% RSLogix 500 project BESTANDMANAGEMENT.RSS, saved by version 8.30.00.16 %
PROJECT "UNTITLED"    % processor: Bul.1763 MicroLogix 1100 Series B %

PROGRAM FILES
  LAD 2 "MAIN"  5 rungs
  LAD 3 "REIFEN"  5 rungs
  LAD 4 "FELGEN"  5 rungs
  LAD 5 "STOßDÄMPFE"  5 rungs

DATA FILES
  O0 OUTPUT  4 elements
  I1 INPUT  6 elements
  S2 STATUS  66 elements
  B3 BINARY  1 elements
  T4 TIMER  1 elements
  C5 COUNTER  1 elements
  R6 CONTROL  1 elements
  N7 INTEGER  9 elements
  F8 FLOAT  1 elements
  ST9 STRING  13 elements

LADDER 2 "MAIN"
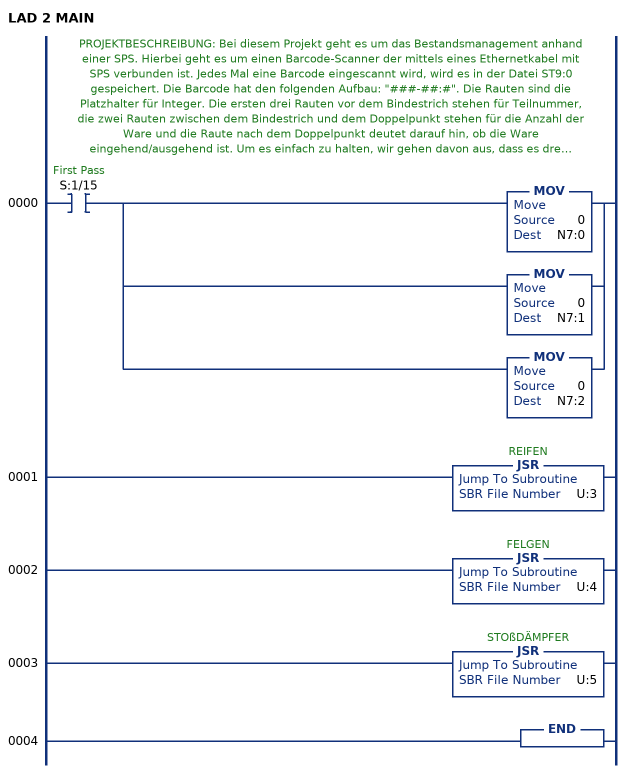
% Rung: 0 %
% PROJEKTBESCHREIBUNG: Bei diesem Projekt geht es um das Bestandsmanagement anhand einer SPS. Hierbei geht es um einen Barcode-Scanner der mittels eines Ethernetkabel mit SPS verbunden ist. Jedes Mal eine Barcode eingescannt wird, wird es in der Datei ST9:0 gespeichert. Die Barcode hat den folgenden Aufbau: "###-##:#". Die Rauten sind die Platzhalter für Integer. Die ersten drei Rauten vor dem Bindestrich stehen für Teilnummer, die zwei Rauten zwischen dem Bindestrich und dem Doppelpunkt stehen für die Anzahl der Ware und die Raute nach dem Doppelpunkt deutet darauf hin, ob die Ware eingehend/ausgehend ist. Um es einfach zu halten, wir gehen davon aus, dass es drei verschiedene Teile verwaltet werden. Teilnummer eins sind die Reifen mit der Teilnummer 123 , Teilnummer zwei sind die Felgen mit der Teilnummer 456 und Teilnummer drei sind die Stoßdämpfer mit der Nummer 789. Die letze Raute ist 1 beim Wareneingang und 2 beim Warenausgang.  N7:0 speichert die Anzahl der Reifen, N7:1 speichert die Anzahl der Felgen und N7:2 speichert die Anzahl der Stoßdämpfer. Beim Initialisierung wird sichergestellt, dass der Lager leer ist. %
SOR XIC S:1/15 BST MOV 0 N7:0 NXB MOV 0 N7:1 NXB MOV 0 N7:2 BND EOR
%   S:1/15  "First Pass" %
% Rung: 1 %
SOR JSR U:3 EOR
%   U:3  "REIFEN" %
% Rung: 2 %
SOR JSR U:4 EOR
%   U:4  "FELGEN" %
% Rung: 3 %
SOR JSR U:5 EOR
%   U:5  "STOßDÄMPFER" %
% Rung: 4 %
SOR END EOR

LADDER 3 "REIFEN"
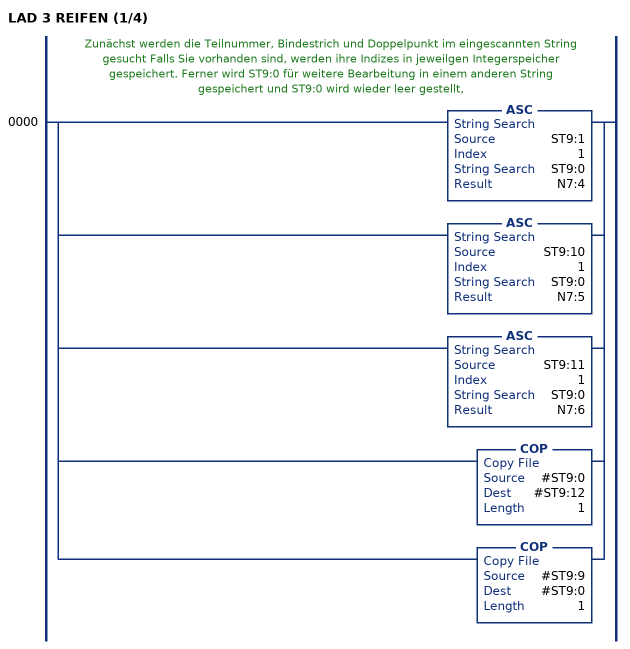
% Rung: 0 %
% Zunächst werden die Teilnummer, Bindestrich und Doppelpunkt im eingescannten String gesucht Falls Sie vorhanden sind, werden ihre Indizes in jeweilgen Integerspeicher gespeichert. Ferner wird ST9:0 für weitere Bearbeitung in einem anderen String gespeichert und ST9:0 wird wieder leer gestellt, %
SOR BST ASC ST9:1 1 ST9:0 N7:4 NXB ASC ST9:10 1 ST9:0 N7:5 NXB ASC ST9:11 1 ST9:0 N7:6 NXB COP #ST9:0 #ST9:12 1 NXB COP #ST9:9 #ST9:0 1 BND EOR
%   N7:4  "Index von Reifennummer" %
%   N7:5  "Index von Bindestrich" %
%   N7:6  "Index von Doppelpunkt" %

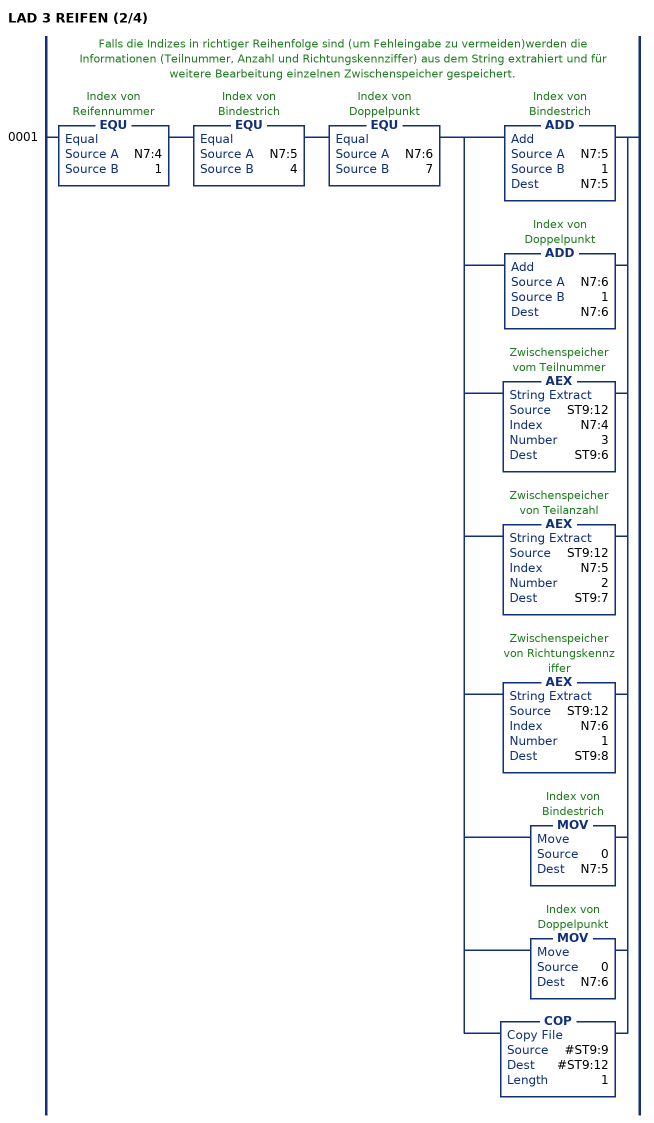
% Rung: 1 %
% Falls die Indizes in richtiger Reihenfolge sind (um Fehleingabe zu vermeiden)werden die Informationen (Teilnummer, Anzahl und Richtungskennziffer) aus dem String extrahiert und für weitere Bearbeitung einzelnen Zwischenspeicher gespeichert. %
SOR EQU N7:4 1 EQU N7:5 4 EQU N7:6 7 BST ADD N7:5 1 N7:5 NXB ADD N7:6 1 N7:6 NXB AEX ST9:12 N7:4 3 ST9:6 NXB AEX ST9:12 N7:5 2 ST9:7 NXB AEX ST9:12 N7:6 1 ST9:8 NXB MOV 0 N7:5 NXB MOV 0 N7:6 NXB COP #ST9:9 #ST9:12 1 BND EOR
%   N7:4  "Index von Reifennummer" %
%   N7:5  "Index von Bindestrich" %
%   N7:6  "Index von Doppelpunkt" %
%   ST9:6  "Zwischenspeicher vom Teilnummer" %
%   ST9:7  "Zwischenspeicher von Teilanzahl" %
%   ST9:8  "Zwischenspeicher von Richtungskennziffer" %

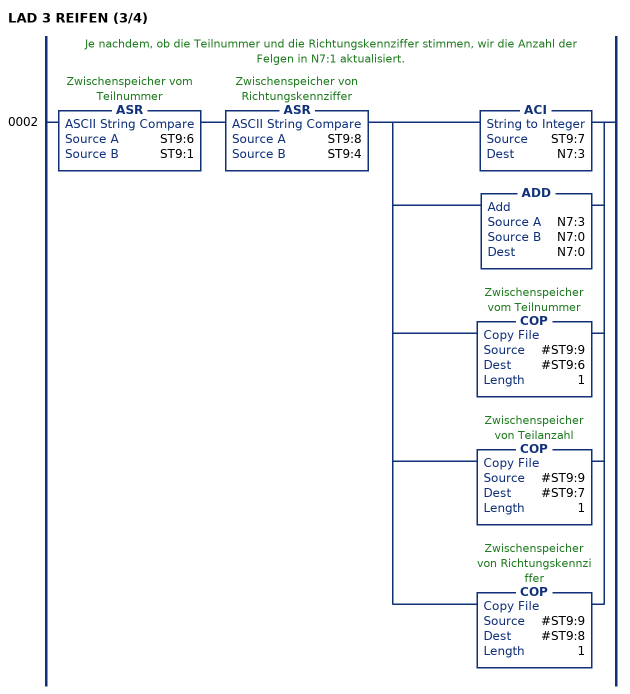
% Rung: 2 %
% Je nachdem, ob die Teilnummer und die Richtungskennziffer stimmen, wir die Anzahl der Felgen in N7:1 aktualisiert. %
SOR ASR ST9:6 ST9:1 ASR ST9:8 ST9:4 BST ACI ST9:7 N7:3 NXB ADD N7:3 N7:0 N7:0 NXB COP #ST9:9 #ST9:6 1 NXB COP #ST9:9 #ST9:7 1 NXB COP #ST9:9 #ST9:8 1 BND EOR
%   ST9:6  "Zwischenspeicher vom Teilnummer" %
%   ST9:8  "Zwischenspeicher von Richtungskennziffer" %
%   ST9:7  "Zwischenspeicher von Teilanzahl" %

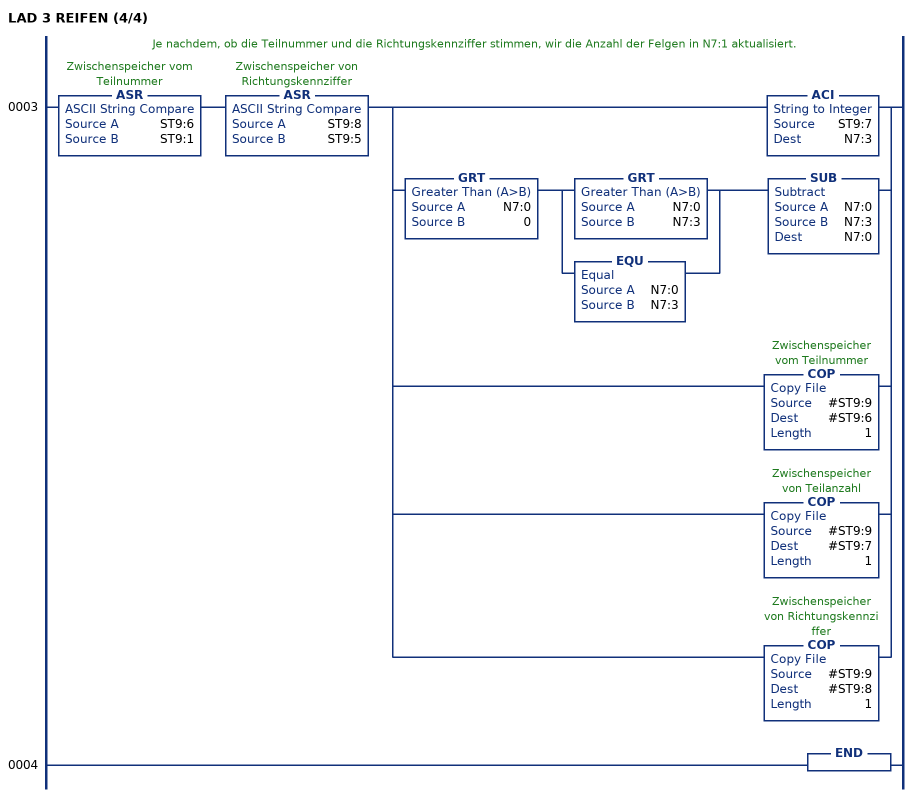
% Rung: 3 %
% Je nachdem, ob die Teilnummer und die Richtungskennziffer stimmen, wir die Anzahl der Felgen in N7:1 aktualisiert. %
SOR ASR ST9:6 ST9:1 ASR ST9:8 ST9:5 BST ACI ST9:7 N7:3 NXB GRT N7:0 0 BST GRT N7:0 N7:3 NXB EQU N7:0 N7:3 BND SUB N7:0 N7:3 N7:0 NXB COP #ST9:9 #ST9:6 1 NXB COP #ST9:9 #ST9:7 1 NXB COP #ST9:9 #ST9:8 1 BND EOR
%   ST9:6  "Zwischenspeicher vom Teilnummer" %
%   ST9:8  "Zwischenspeicher von Richtungskennziffer" %
%   ST9:7  "Zwischenspeicher von Teilanzahl" %
% Rung: 4 %
SOR END EOR

LADDER 4 "FELGEN"
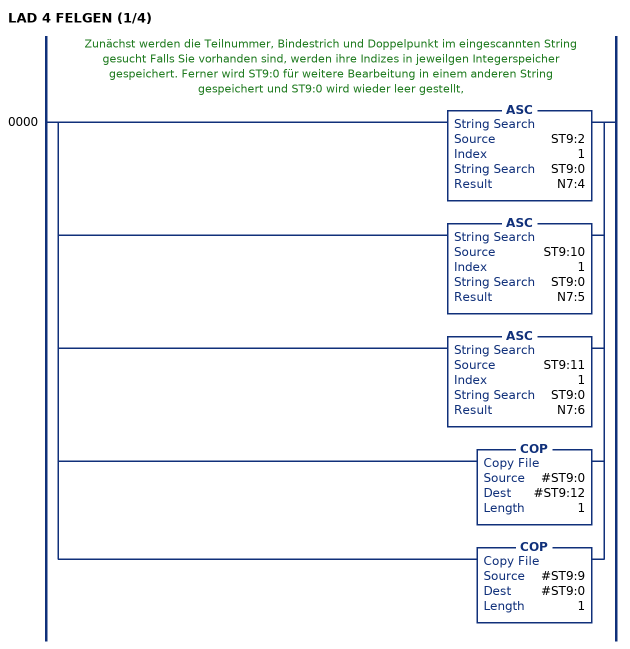
% Rung: 0 %
% Zunächst werden die Teilnummer, Bindestrich und Doppelpunkt im eingescannten String gesucht Falls Sie vorhanden sind, werden ihre Indizes in jeweilgen Integerspeicher gespeichert. Ferner wird ST9:0 für weitere Bearbeitung in einem anderen String gespeichert und ST9:0 wird wieder leer gestellt, %
SOR BST ASC ST9:2 1 ST9:0 N7:4 NXB ASC ST9:10 1 ST9:0 N7:5 NXB ASC ST9:11 1 ST9:0 N7:6 NXB COP #ST9:0 #ST9:12 1 NXB COP #ST9:9 #ST9:0 1 BND EOR
%   N7:4  "Index von Reifennummer" %
%   N7:5  "Index von Bindestrich" %
%   N7:6  "Index von Doppelpunkt" %

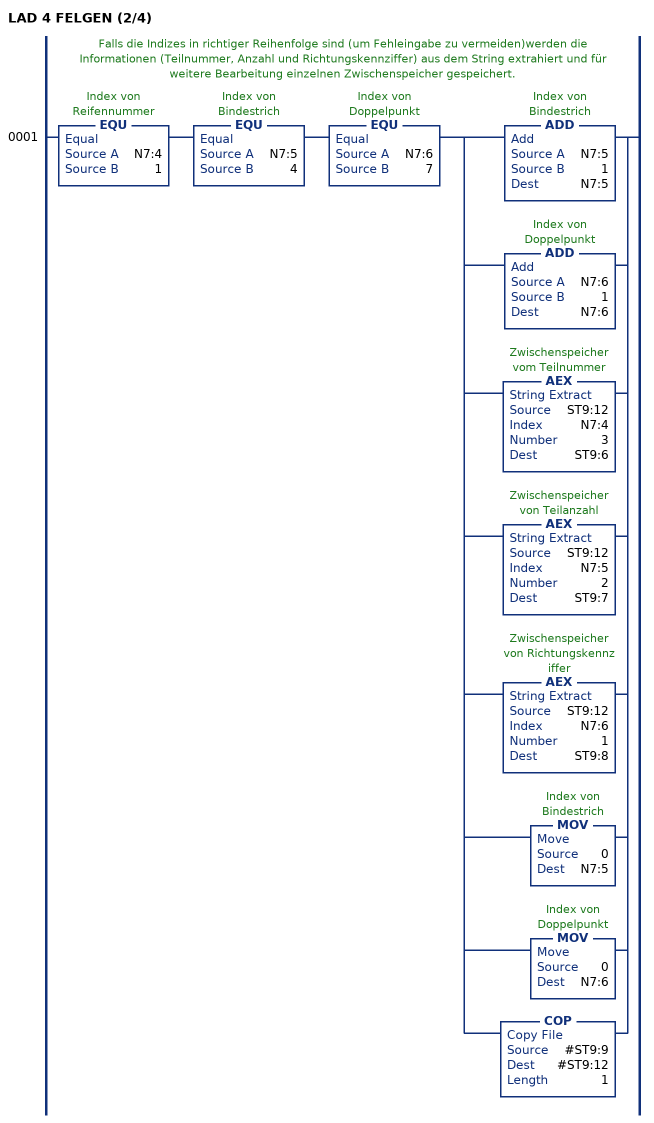
% Rung: 1 %
% Falls die Indizes in richtiger Reihenfolge sind (um Fehleingabe zu vermeiden)werden die Informationen (Teilnummer, Anzahl und Richtungskennziffer) aus dem String extrahiert und für weitere Bearbeitung einzelnen Zwischenspeicher gespeichert. %
SOR EQU N7:4 1 EQU N7:5 4 EQU N7:6 7 BST ADD N7:5 1 N7:5 NXB ADD N7:6 1 N7:6 NXB AEX ST9:12 N7:4 3 ST9:6 NXB AEX ST9:12 N7:5 2 ST9:7 NXB AEX ST9:12 N7:6 1 ST9:8 NXB MOV 0 N7:5 NXB MOV 0 N7:6 NXB COP #ST9:9 #ST9:12 1 BND EOR
%   N7:4  "Index von Reifennummer" %
%   N7:5  "Index von Bindestrich" %
%   N7:6  "Index von Doppelpunkt" %
%   ST9:6  "Zwischenspeicher vom Teilnummer" %
%   ST9:7  "Zwischenspeicher von Teilanzahl" %
%   ST9:8  "Zwischenspeicher von Richtungskennziffer" %

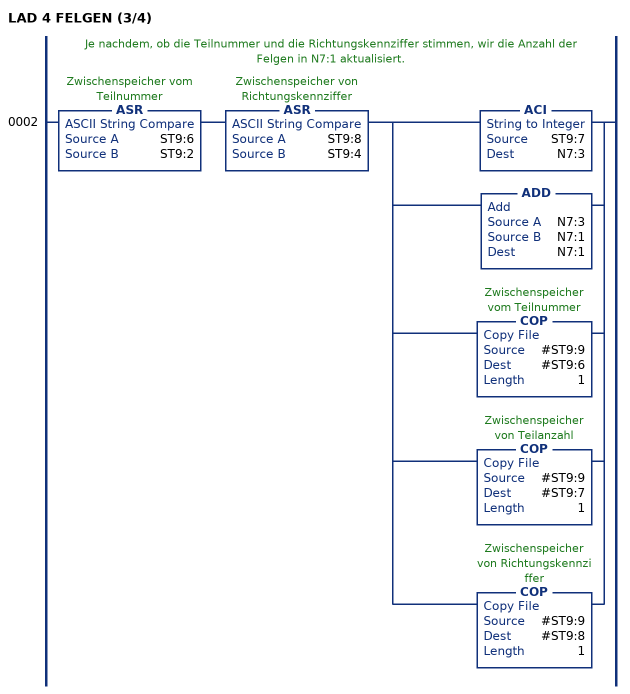
% Rung: 2 %
% Je nachdem, ob die Teilnummer und die Richtungskennziffer stimmen, wir die Anzahl der Felgen in N7:1 aktualisiert. %
SOR ASR ST9:6 ST9:2 ASR ST9:8 ST9:4 BST ACI ST9:7 N7:3 NXB ADD N7:3 N7:1 N7:1 NXB COP #ST9:9 #ST9:6 1 NXB COP #ST9:9 #ST9:7 1 NXB COP #ST9:9 #ST9:8 1 BND EOR
%   ST9:6  "Zwischenspeicher vom Teilnummer" %
%   ST9:8  "Zwischenspeicher von Richtungskennziffer" %
%   ST9:7  "Zwischenspeicher von Teilanzahl" %

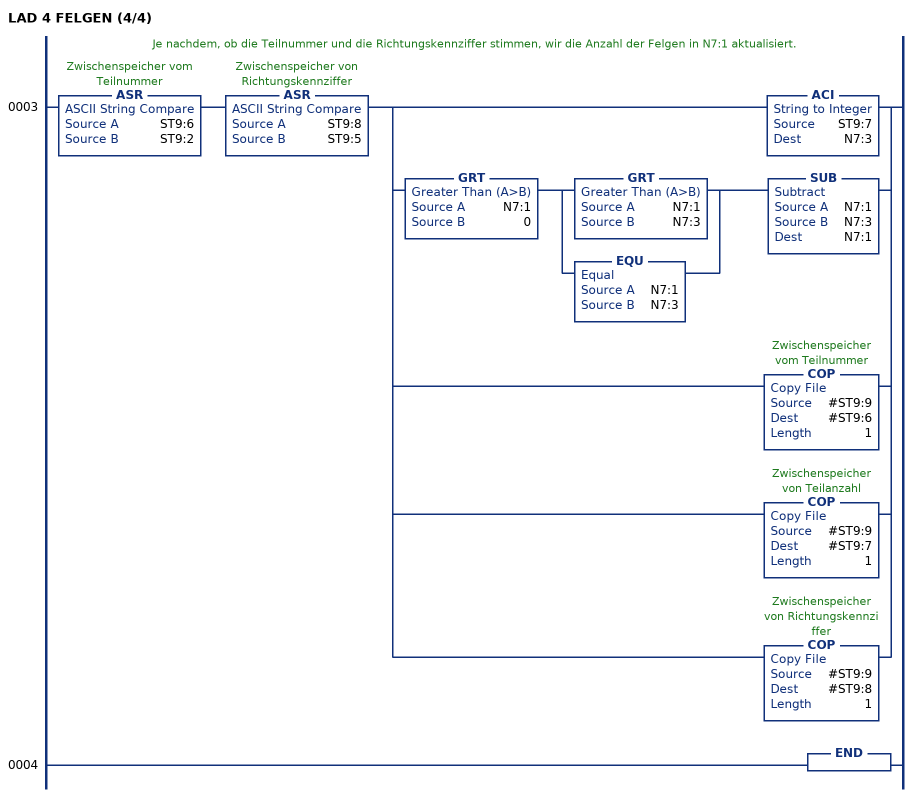
% Rung: 3 %
% Je nachdem, ob die Teilnummer und die Richtungskennziffer stimmen, wir die Anzahl der Felgen in N7:1 aktualisiert. %
SOR ASR ST9:6 ST9:2 ASR ST9:8 ST9:5 BST ACI ST9:7 N7:3 NXB GRT N7:1 0 BST GRT N7:1 N7:3 NXB EQU N7:1 N7:3 BND SUB N7:1 N7:3 N7:1 NXB COP #ST9:9 #ST9:6 1 NXB COP #ST9:9 #ST9:7 1 NXB COP #ST9:9 #ST9:8 1 BND EOR
%   ST9:6  "Zwischenspeicher vom Teilnummer" %
%   ST9:8  "Zwischenspeicher von Richtungskennziffer" %
%   ST9:7  "Zwischenspeicher von Teilanzahl" %
% Rung: 4 %
SOR END EOR

LADDER 5 "STOßDÄMPFE"
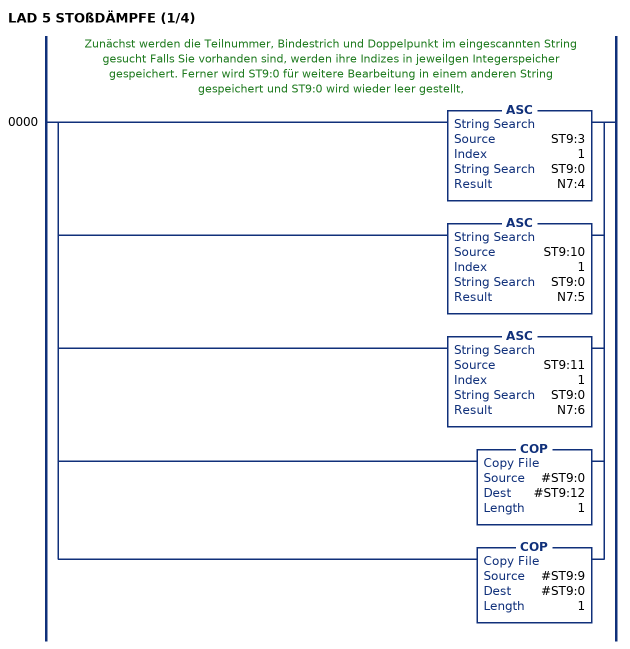
% Rung: 0 %
% Zunächst werden die Teilnummer, Bindestrich und Doppelpunkt im eingescannten String gesucht Falls Sie vorhanden sind, werden ihre Indizes in jeweilgen Integerspeicher gespeichert. Ferner wird ST9:0 für weitere Bearbeitung in einem anderen String gespeichert und ST9:0 wird wieder leer gestellt, %
SOR BST ASC ST9:3 1 ST9:0 N7:4 NXB ASC ST9:10 1 ST9:0 N7:5 NXB ASC ST9:11 1 ST9:0 N7:6 NXB COP #ST9:0 #ST9:12 1 NXB COP #ST9:9 #ST9:0 1 BND EOR
%   N7:4  "Index von Reifennummer" %
%   N7:5  "Index von Bindestrich" %
%   N7:6  "Index von Doppelpunkt" %

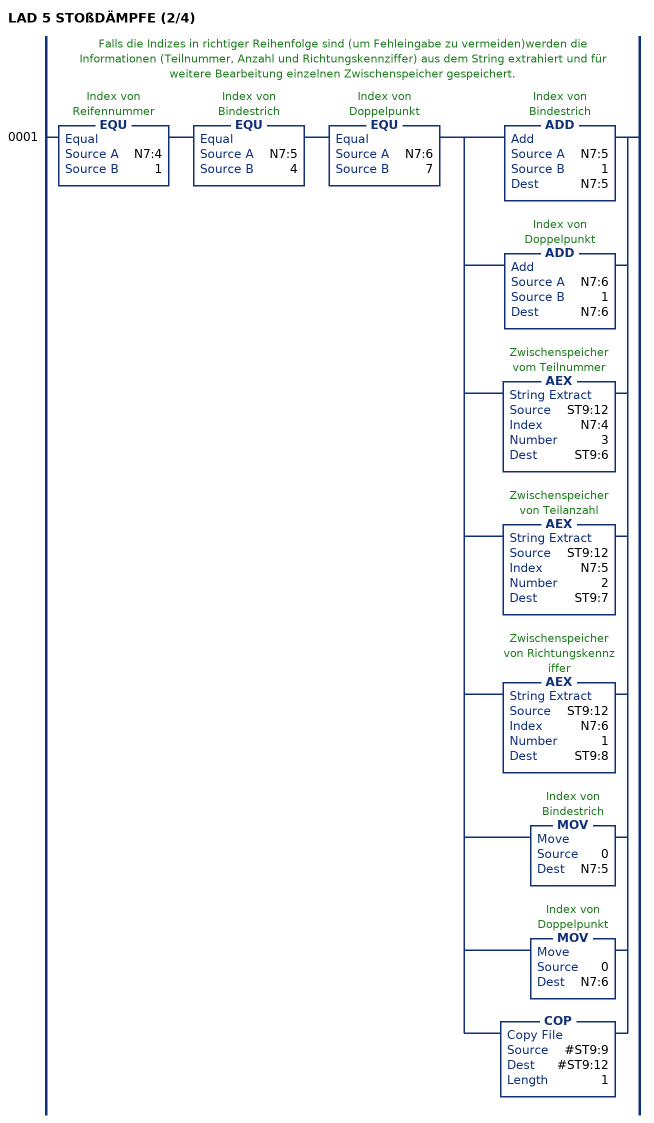
% Rung: 1 %
% Falls die Indizes in richtiger Reihenfolge sind (um Fehleingabe zu vermeiden)werden die Informationen (Teilnummer, Anzahl und Richtungskennziffer) aus dem String extrahiert und für weitere Bearbeitung einzelnen Zwischenspeicher gespeichert. %
SOR EQU N7:4 1 EQU N7:5 4 EQU N7:6 7 BST ADD N7:5 1 N7:5 NXB ADD N7:6 1 N7:6 NXB AEX ST9:12 N7:4 3 ST9:6 NXB AEX ST9:12 N7:5 2 ST9:7 NXB AEX ST9:12 N7:6 1 ST9:8 NXB MOV 0 N7:5 NXB MOV 0 N7:6 NXB COP #ST9:9 #ST9:12 1 BND EOR
%   N7:4  "Index von Reifennummer" %
%   N7:5  "Index von Bindestrich" %
%   N7:6  "Index von Doppelpunkt" %
%   ST9:6  "Zwischenspeicher vom Teilnummer" %
%   ST9:7  "Zwischenspeicher von Teilanzahl" %
%   ST9:8  "Zwischenspeicher von Richtungskennziffer" %

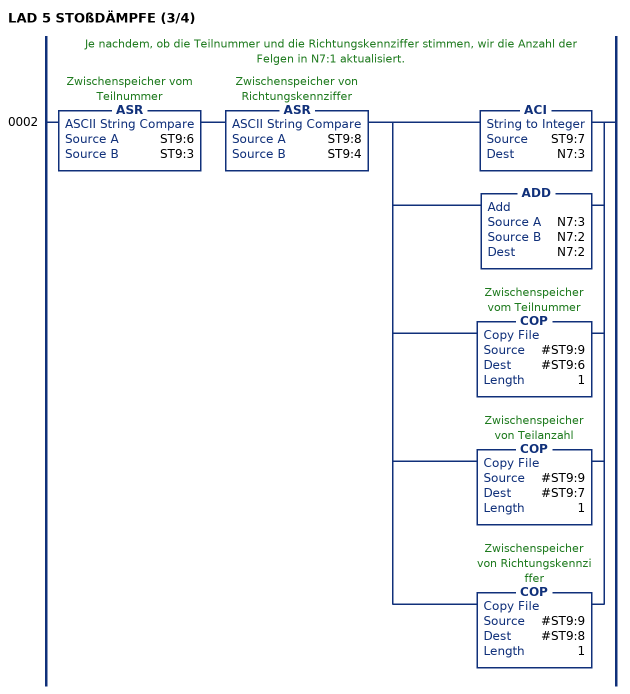
% Rung: 2 %
% Je nachdem, ob die Teilnummer und die Richtungskennziffer stimmen, wir die Anzahl der Felgen in N7:1 aktualisiert. %
SOR ASR ST9:6 ST9:3 ASR ST9:8 ST9:4 BST ACI ST9:7 N7:3 NXB ADD N7:3 N7:2 N7:2 NXB COP #ST9:9 #ST9:6 1 NXB COP #ST9:9 #ST9:7 1 NXB COP #ST9:9 #ST9:8 1 BND EOR
%   ST9:6  "Zwischenspeicher vom Teilnummer" %
%   ST9:8  "Zwischenspeicher von Richtungskennziffer" %
%   ST9:7  "Zwischenspeicher von Teilanzahl" %

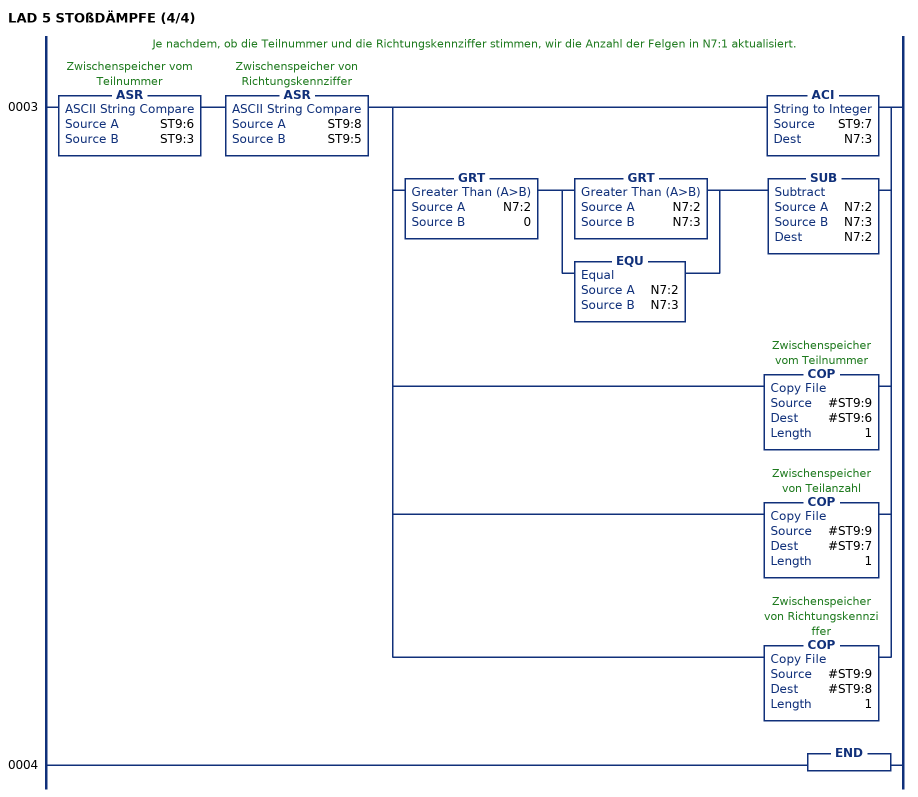
% Rung: 3 %
% Je nachdem, ob die Teilnummer und die Richtungskennziffer stimmen, wir die Anzahl der Felgen in N7:1 aktualisiert. %
SOR ASR ST9:6 ST9:3 ASR ST9:8 ST9:5 BST ACI ST9:7 N7:3 NXB GRT N7:2 0 BST GRT N7:2 N7:3 NXB EQU N7:2 N7:3 BND SUB N7:2 N7:3 N7:2 NXB COP #ST9:9 #ST9:6 1 NXB COP #ST9:9 #ST9:7 1 NXB COP #ST9:9 #ST9:8 1 BND EOR
%   ST9:6  "Zwischenspeicher vom Teilnummer" %
%   ST9:8  "Zwischenspeicher von Richtungskennziffer" %
%   ST9:7  "Zwischenspeicher von Teilanzahl" %
% Rung: 4 %
SOR END EOR

COMMENTS NOT ATTACHED TO A CURRENT RUNG
  ST9:11: Das Program startet mit der Suche von Teilnummer und speichert den Index von String, bei dem es die Teilnummer findet, in N7:4. In den nächsten beiden Schritten werden die Indizes vom Bindestrich und Doppelpunkt gesucht und werden in jeweiligen Plätze als Integer gespeichert.

DATA TABLE (non-zero values as saved)
DATA N7
% N7:0 % 40 0 0 60 1 0 0 8 5
DATA ST9
% ST9:1 % "123"
% ST9:2 % "456"
% ST9:3 % "789"
% ST9:4 % "1"
% ST9:5 % "2"
% ST9:7 % "60"
% ST9:10 % "-"
% ST9:11 % ":"
